FUNCTION_BLOCK sftDiCondAck
VAR
END_VAR
VAR_INPUT
	mcbutB1:=sftDiModule.sftDiRunVE1;
	mcbutB2:=sftDiModule.sftDiRunVE2;
	mcbutB3:=sftDiModule.sftDiRunVE3;
	mcbutB4:=sftDiModule.sftDiRunVE4;
END_VAR
VAR
END_VAR
VAR_OUTPUT
	sentREF1: BOOL;
	sentREF2: BOOL;
	sentREF3: BOOL;
	sentREF4: BOOL;
END_VAR
VAR
END_VAR

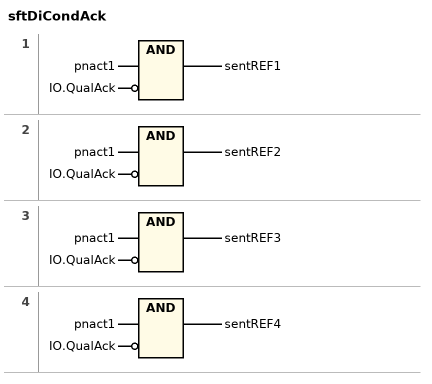
// NETWORK 1
sentREF1 := pnact1 AND NOT IO.QualAck;

// NETWORK 2
sentREF2 := pnact1 AND NOT IO.QualAck;

// NETWORK 3
sentREF3 := pnact1 AND NOT IO.QualAck;

// NETWORK 4
sentREF4 := pnact1 AND NOT IO.QualAck;

END_FUNCTION_BLOCK

(* stored: Version 1.1.0.1, ProductVersion 3.1.4024.0
   POU sftDiCondAck: Id {2b2c26fc-df07-4d92-bb82-ffc58ea04212}, SpecialFunc None *)
